FUNCTION_BLOCK _FB_BufferWriter
VAR_INPUT
	pRawBuf : POINTER TO BYTE; 
	nSize : UDINT;
END_VAR

VAR_OUTPUT
	nCurOffset : UDINT;
END_VAR

VAR
END_VAR

METHOD SetOffset : BOOL
VAR_INPUT
	nOffset : UDINT;
END_VAR
IF nOffset >= nSize THEN
	SetOffset := FALSE;
ELSE
	nCurOffset := nOffset;	
	SetOffset := TRUE;
END_IF
END_METHOD

METHOD Write : BOOL
VAR_INPUT
	pSrc : POINTER TO BYTE;
	nBytes : UDINT;
END_VAR
IF nCurOffset + nBytes >= nSize THEN
	Write := FALSE;
ELSE
	Write := SAFE_MEMCPY(ADR(pRawBuf[nCurOffset]), nSize, pSrc, nBytes);
	nCurOffset := nCurOffset + nBytes;	
END_IF
END_METHOD

METHOD WriteAt : BOOL
VAR_INPUT
	nIndex : UDINT;
	pSrc : POINTER TO BYTE;
	nBytes : UDINT;
END_VAR
WriteAt := SAFE_MEMCPY(ADR(pRawBuf[nIndex]), nSize-nIndex, pSrc, nBytes);
END_METHOD

METHOD WriteByte : BOOL
VAR_INPUT
	nByte : BYTE;
END_VAR
IF nCurOffset < nSize THEN
	pRawBuf[nCurOffset] := nByte;
	nCurOffset := nCurOffset + 1;
	WriteByte := TRUE;
ELSE
	WriteByte := FALSE;
END_IF
END_METHOD

END_FUNCTION_BLOCK

(* stored: Version 1.1.0.1
   POU _FB_BufferWriter: Id {f3d5358a-0bf2-4a52-9f95-9801ddb8841e}, SpecialFunc None
   Method SetOffset: Id {073d1dd1-b5f7-4f4f-8f3e-dfd435173099}
   Method Write: Id {eff76194-79d9-4d9c-9b14-16156e53c9eb}
   Method WriteAt: Id {b0c2235a-a289-49c6-8e22-f373296a49a0}
   Method WriteByte: Id {83829bc1-d501-4035-a0f9-a6d297ae4b16} *)
